// Mitsubishi GX Works2 project: 240416_지연동작한시복귀   PLC: Q03UDV

PROGRAM MAIN
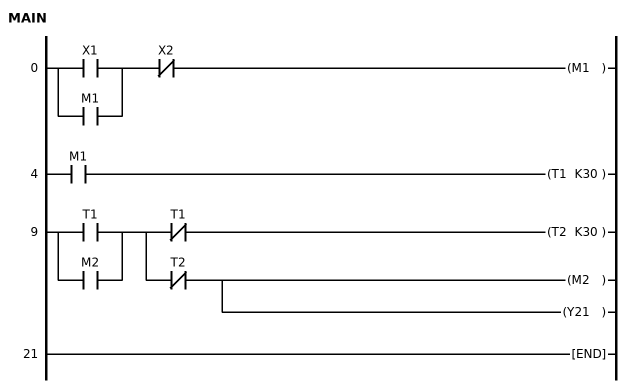
0     LD      X1
      OR      M1
      ANI     X2
      OUT     M1
4     LD      M1
      OUT     T1 K30
9     LD      T1
      OR      M2
      MPS
      ANI     T1
      OUT     T2 K30
      MPP
      ANI     T2
      OUT     M2
      OUT     Y21
21    END
END_PROGRAM
